(* IEC 61131-3 sources: programs/VI-54/VI-54_20171205/VI-54_20171205/Stations/Screen/LseClass170718/Class/SaveLoadUSB, 1 file *)

(* ---- SaveLoadUSB.st ---- *)
(*!
<Class
	Name               = "SaveLoadUSB"
	Revision           = "0.0"
	RealtimeTask       = "false"
	CyclicTask         = "false"
	BackgroundTask     = "false"
	Sigmatek           = "false"
	OSInterface        = "false"
	HighPriority       = "false"
	Automatic          = "false"
	UpdateMode         = "Prescan"
	SharedCommandTable = "true"
	Objectsize         = "(540,540)">
	<Channels>
		<Server Name="Copy" Visualized="true" Initialize="false" WriteProtected="false" Retentive="false"/>
		<Server Name="ResultFileCopy" Visualized="false" Initialize="false" WriteProtected="true" Retentive="false"/>
		<Server Name="UserUSBLinked" Visualized="true" Initialize="false" WriteProtected="true" Retentive="false"/>
		<Client Name="FileOs" Required="false" Internal="false"/>
		<Client Name="System" Required="false" Internal="false"/>
		<Client Name="vLevel" Required="true" Internal="false"/>
	</Channels>
	<Network Name="SaveLoadUSB">
		<!-- List of Components in this network -->
		<Components>
			<Object
				Name       = "_base"
				Class      = "_Global"
				Position   = "(218,120)"
				Visualized = "true"
				Remotely   = "true">
				<Channels>
					<Server Name="Server0"/>
					<Client Name="Lse"/>
				</Channels>
			</Object>
		</Components>
		<Comments>
		</Comments>
		<!-- List of Connections in this network -->
		<Connections>
			<Connection Source="this.Server0" Destination="_base.Server0" Vertices="(690,210),(518,210),"/>
			<Connection Source="_base.Lse" Destination="this.Lse" Vertices="(218,210),(38,210),"/>
		</Connections>
		<!-- Headerfiles -->
		<Options>
		</Options>
	</Network>
</Class>
*)
#pragma using _Global

SaveLoadUSB : CLASS
: _Global
	TYPE
	  CharArray : ARRAY [0..100] OF CHAR;
	END_TYPE
  //Servers:
	Copy 	: SvrCh_DINT;
	ResultFileCopy 	: SvrCh_DINT;
	UserUSBLinked 	: SvrCh_DINT;
  //Clients:
	FileOs 	: CltChCmd__FileSys;
	System 	: CltChCmd_System;
	vLevel 	: CltCh_DINT;
  //Variables:
		CodeOk 	: DINT;
  //Functions:

	FUNCTION VIRTUAL GLOBAL Init;

	FUNCTION VIRTUAL GLOBAL IF_WindowRun
		VAR_INPUT
			whoami 	: ^_WHOAMI;
			pic 	: ^void;
			event 	: ^_EVENT;
		END_VAR;

	FUNCTION VIRTUAL GLOBAL Copy::Write
		VAR_INPUT
			input (EAX) 	: DINT;
		END_VAR
		VAR_OUTPUT
			result (EAX) 	: DINT;
		END_VAR;
  //Tables:
	FUNCTION @STD
		VAR_OUTPUT
			ret_code	: CONFSTATES;
		END_VAR;
	FUNCTION GLOBAL TAB @CT_;
END_CLASS;

#pragma usingLtd _FileSys
#pragma usingLtd System

FUNCTION VIRTUAL GLOBAL SaveLoadUSB::Init

  //call method from base class
  _Global::init();

  if _firstscan = 1 then
//    DiskSpace := FileOs.GetDiskSpace(Drive:="c", BytesPerSector:=512, SectorsPerCluster:=, TotalClusters:=, FreeClusters:=);
  end_if;

END_FUNCTION

FUNCTION VIRTUAL GLOBAL SaveLoadUSB::IF_WindowRun
	VAR_INPUT
		whoami 	: ^_WHOAMI;
		pic 	: ^void;
		event 	: ^_EVENT;
	END_VAR

    //call method from baseclass
  _Global::IF_WindowRun(whoami, pic, event);

  if event^.ftype <> _EVENT_NONE then
    //Check if there is some action on the usb-port
    if ( event^.ftype = _EVENT_LASALOS ) & ( event^.scancode = 8 )then
      if event^.modifier = 1 then
        UserUSBLinked := 1;
      elsif event^.modifier = 2 then
        UserUSBLinked := 0;
      end_if;
    end_if;
  end_if;

  // check code..
  if IsClientConnected(#vLevel ) then
    vLevel := vLevel.Read();
  end_if;

  // bij juiste level is saven ook mogelijk
  if vLevel >= TECHNICIAN then
    CodeOk := 1;
  else
    CodeOk := 0;
  end_if;

  case Copy of
    00:

    01:// from ETV to USB (eventjournaal)
      if CodeOk = 1 then
        if FileOs.CreateDirectory(dirname:= "E:\eventjournal") >= 0 then  // "c:\product\*.csv"
          Copy += 1; //
        else
          Copy += 1; //   can't make dir. (dir already exsist)
        end_if;
      end_if;
    02: // copy EventJournaal
      ResultFileCopy := FileOs.FileCopy(pSource:="C:\export\eventjournal", pDest:= "E:\eventjournal", udOption := FC_SUBDIRECTORIES);
      Copy := 0;

    10:// from ETV to USB (toolcat)
      if CodeOk = 1 then
        if FileOs.CreateDirectory(dirname:= "E:\Toolcat") >= 0 then  // "c:\product\*.csv"
          Copy += 1; //
        else
          Copy += 1; //   can't make dir. (dir already exsist)
        end_if;
      end_if;
    11: // copy
      ResultFileCopy := FileOs.FileCopy(pSource:="c:\Toolcat", pDest:= "E:\Toolcat", udOption := FC_SUBDIRECTORIES);
      Copy := 0;

    14:// From USB to ETV (toolcat)
      if CodeOk = 1 then
        if FileOs.CreateDirectory(dirname:="C:\Toolcat") >= 0 then
          Copy += 1; //
        else
          Copy += 1; //   can't make dir.(dir already exsist)
        end_if;
      end_if;
    15:
      ResultFileCopy := FileOs.FileCopy(pSource:="E:\Toolcat", pDest:= "C:\Toolcat", udOption := FC_SUBDIRECTORIES);
      Copy := 0;

    20:// from ETV to USB (SpareParts)
      if CodeOk = 1 then
        if FileOs.CreateDirectory(dirname:= "E:\Spareparts") >= 0 then  // "c:\product\*.csv"
          Copy += 1; //
        else
          Copy += 1; //   can't make dir. (dir already exsist)
        end_if;
      end_if;
    21: // copy
      ResultFileCopy := FileOs.FileCopy(pSource:="c:\Spareparts", pDest:= "E:\Spareparts", udOption := FC_SUBDIRECTORIES);
      Copy := 0;

    24:// From USB to ETV (SpareParts)
      if CodeOk = 1 then
        if FileOs.CreateDirectory(dirname:="C:\Spareparts") >= 0 then
          Copy += 1; //
        else
          Copy += 1; //   can't make dir.(dir already exsist)
        end_if;
      end_if;
    25:
      ResultFileCopy := FileOs.FileCopy(pSource:="E:\Spareparts", pDest:= "C:\Spareparts", udOption := FC_SUBDIRECTORIES);
      Copy := 0;
  end_case;

END_FUNCTION
FUNCTION VIRTUAL GLOBAL SaveLoadUSB::Copy::Write
	VAR_INPUT
		input (EAX) 	: DINT;
	END_VAR
	VAR_OUTPUT
		result (EAX) 	: DINT;
	END_VAR

	Copy := input;
 	result := Copy;

END_FUNCTION
